TYPE T_Ctrl_Alm :
STRUCT
	///alarm flag array
	bol: BOOL;
	eAlmClass: E_AlmClass;
	strText: STRING;
END_STRUCT
END_TYPE

(* stored: Version 1.1.0.1, ProductVersion 3.1.0.18
   DUT T_Ctrl_Alm: Id {cd2bbfb8-56c1-4c3e-ad1d-cc225e01ab34} *)
